TYPE LED1904 :
STRUCT
	bInput1:BOOL;
	bInput2:BOOL;
	bInput3:BOOL;
	bInput4:BOOL;
	bDiag1:BOOL;
	bDiag2:BOOL;
	bDiag3:BOOL;
	bDiag4:BOOL;
END_STRUCT
END_TYPE

(* stored: Version 1.1.0.1, ProductVersion 3.1.4024.12
   DUT LED1904: Id {4661467b-3c66-4bf8-b569-6f4f09352f51} *)
